PROGRAM Test
VAR
END_VAR

// NETWORK 1

END_PROGRAM

(* stored: Version 1.1.0.1, ProductVersion 3.1.4026.13
   POU Test: Id {c73af5e4-5324-4b0d-a72b-e19036e19588}, SpecialFunc None *)
